// TIA Portal V18 export
DATA_BLOCK "ST10_PM"   // DB1063
{ S7_Optimized_Access := 'FALSE' }
// stored: AutoNumber false
   VAR RETAIN
      Num : Array[1..32] of "RCS_PMInterface_V1";
      Status { S7_SetPoint := 'True'} : Array[1..50] of Int;
   END_VAR
BEGIN
   // Num[1] : laszer marking
   // Num[2] : LabelFeeder
END_DATA_BLOCK
